(* PLC project CHL-DZ-BJDX-11 宁波数字孪生（东方理工）研究院制备薄层色谱全自动化工作站_Old_InoProShop(V1.9.1.6).project, Inovance company InoProShop(V1.9.1.6) InoProShop(V1.9.1.6) *)
(* stored: creationDateTime 2026-06-16T17:57:29.9700021, modificationDateTime 2026-06-04T10:59:46 *)

PROGRAM initialization

            上样轴4X轴DATE.bHomed:=FALSE;
上样轴5Z轴DATE.bHomed:=FALSE;
          
END_PROGRAM
